(* IEC 61131-3 sources: eCockpitGit/test_project/src/%F%00 Library/%F%Common Functions/%F%Networking, 7 files *)

(* ---- %POU%BASE64Decode.st ---- *)
//This function decodes a base64 string to a normal string or byte array
// |**Version**|**Author**| **Date** |**Changes**
// | 1         | NSN      | 19-05-20 | Creation
FUNCTION BASE64Decode : BOOL
VAR_INPUT
	inStr		:POINTER TO BYTE;
	outStr		:POINTER TO BYTE;		//Out string must be at least 3/4 as long as input string and also a multiple of 4
END_VAR
VAR
	inStrNext	:POINTER TO BYTE := inStr + 1;
	baseBuffer	:BYTE;
END_VAR
VAR CONSTANT
	base64Vars	:ARRAY[43..122] OF BYTE := [62,0,0,0,63,52,53,54,55,56,57,58,59,60,61,0,0,0,0,0,0,0,0,1,2,3,4,5,6,7,8,9,10,11,12,13,14,15,16,17,18,19,20,21,22,23,24,25,0,0,0,0,0,0,26,27,28,29,30,31,32,33,34,35,36,37,38,39,40,41,42,43,44,45,46,47,48,49,50,51];
END_VAR

(*%!%__DELIMITER__%!%*)
WHILE inStr^ <> 0 AND inStrNext^ <> 0 DO
	baseBuffer				:=		SHL(base64Vars[inStr^],2) OR SHR(base64Vars[inStrNext^],4);
	outStr^					:=		baseBuffer;
	inStr					:=		inStr + 1;
	inStrNext				:=		inStr + 1;
	outStr					:=		outStr + 1;
	IF inStr^ <> 0 AND inStrNext^ <> 0 THEN
		baseBuffer			:=		SHL(base64Vars[inStr^],4) OR SHR(base64Vars[inStrNext^],2);
		outStr^				:=		baseBuffer;
		inStr				:=		inStr + 1;
		inStrNext			:=		inStr + 1;
		outStr				:=		outStr + 1;
		IF inStr^ <> 0 AND inStrNext^ <> 0 THEN
			baseBuffer		:=		SHL(base64Vars[inStr^],6) OR base64Vars[inStrNext^];
			outStr^			:=		baseBuffer;
			inStr			:=		inStr + 2;
			inStrNext		:=		inStr + 1;
			outStr			:=		outStr + 1;
		END_IF
	END_IF
END_WHILE

(* ---- %POU%BASE64Encode.st ---- *)
//This function encodes a normal string or byte array to a base 64 string
// |**Version**|**Author**| **Date** |**Changes**
// | 1         | NSN      | 19-05-20 | Creation
FUNCTION BASE64Encode : BOOL
VAR_INPUT
	inStr		:POINTER TO BYTE;		//Input string
	outStr		:POINTER TO BYTE;		//Out string must be at least 1/3 longer than input string and also a multiple of 4
END_VAR
VAR
	inStrLast	:POINTER TO BYTE := inStr;
END_VAR
VAR CONSTANT
	base64Vars	:ARRAY[0..63] OF BYTE := [65,66,67,68,69,70,71,72,73,74,75,76,77,78,79,80,81,82,83,84,85,86,87,88,89,90,97,98,99,100,101,102,103,104,105,106,107,108,109,110,111,112,113,114,115,116,117,118,119,120,121,122,48,49,50,51,52,53,54,55,56,57,43,47];
END_VAR

(*%!%__DELIMITER__%!%*)
WHILE inStr^ <> 0 DO
	outStr^					:=		base64Vars[SHR(inStr^,2)];
	inStrLast				:=		inStr;
	inStr					:=		inStr + 1;
	outStr					:=		outStr + 1;
	IF inStr^ = 0 THEN
		outStr^				:=		base64Vars[SHR(inStr^,4) OR SHL(inStrLast^,4) AND 63];
		outStr				:=		outStr + 1;
		outStr^				:=		EASCII.Equal;
		outStr				:=		outStr + 1;
		outStr^				:=		EASCII.Equal;
	ELSE
		outStr^				:=		base64Vars[SHR(inStr^,4) OR SHL(inStrLast^,4) AND 63];
		inStrLast			:=		inStr;
		outStr				:=		outStr + 1;
		inStr				:=		inStr + 1;
		IF inStr^ = 0 AND inStrLast^ = 0 THEN
			outStr^			:=		EASCII.Equal;
			outStr			:=		outStr + 1;
			outStr^			:=		EASCII.Equal;
		ELSE
			outStr^			:=		base64Vars[SHR(inStr^,6) OR SHL(inStrLast^,2) AND 63];
			outStr			:=		outStr + 1;
			IF inStr^ = 0 THEN
				outStr^		:=		EASCII.Equal;
			ELSE
				outStr^		:=		base64Vars[inStr^ AND 63];
				outStr		:=		outStr + 1;
				inStr		:=		inStr + 1;
			END_IF
		END_IF
	END_IF
END_WHILE
outStr						:=		outStr + 1;
outStr^						:=		0;

(* ---- %POU%BASE64EncodeLen.st ---- *)
//This function encodes a normal string or byte array of fixed lenght to a base 64 string
//This version exists to process strings with zeros in them
// |**Version**|**Author**| **Date** |**Changes**
// | 1         | NSN      | 19-05-20 | Creation
FUNCTION BASE64EncodeLen : BOOL
VAR_INPUT
	inStr		:POINTER TO BYTE;		//Input string
	inLen		:WORD;					//Lenght of input string
	outStr		:POINTER TO BYTE;		//Out string must be at least 1/3 longer than input string and also a multiple of 4
END_VAR
VAR
	inStrLast	:POINTER TO BYTE := inStr;
END_VAR
VAR CONSTANT
	base64Vars	:ARRAY[0..63] OF BYTE := [65,66,67,68,69,70,71,72,73,74,75,76,77,78,79,80,81,82,83,84,85,86,87,88,89,90,97,98,99,100,101,102,103,104,105,106,107,108,109,110,111,112,113,114,115,116,117,118,119,120,121,122,48,49,50,51,52,53,54,55,56,57,43,47];
END_VAR

(*%!%__DELIMITER__%!%*)
WHILE inLen > 0 DO
	outStr^					:=		base64Vars[SHR(inStr^,2)];
	inStrLast				:=		inStr;
	inStr					:=		inStr + 1;
	outStr					:=		outStr + 1;
	inLen					:=		inLen - 1;
	IF inLen = 0 THEN
		outStr^				:=		base64Vars[SHR(0,4) OR SHL(inStrLast^,4) AND 63];
		outStr				:=		outStr + 1;
		outStr^				:=		EASCII.Equal;
		outStr				:=		outStr + 1;
		outStr^				:=		EASCII.Equal;
	ELSE
		outStr^				:=		base64Vars[SHR(inStr^,4) OR SHL(inStrLast^,4) AND 63];
		inStrLast			:=		inStr;
		outStr				:=		outStr + 1;
		inStr				:=		inStr + 1;
		IF inLen = 1 THEN
			outStr^			:=		base64Vars[SHR(0,6) OR SHL(inStrLast^,2) AND 63];
			outStr			:=		outStr + 1;
			outStr^			:=		EASCII.Equal;
			inLen			:=		inLen - 1;
		ELSE
			outStr^			:=		base64Vars[SHR(inStr^,6) OR SHL(inStrLast^,2) AND 63];
			outStr			:=		outStr + 1;
			inLen			:=		inLen - 1;
			IF inLen = 0 THEN
				outStr^		:=		EASCII.Equal;
			ELSE
				outStr^		:=		base64Vars[inStr^ AND 63];
				outStr		:=		outStr + 1;
				inStr		:=		inStr + 1;
				inLen		:=		inLen - 1;
			END_IF
		END_IF
	END_IF
END_WHILE
outStr						:=		outStr + 1;
outStr^						:=		0;

(* ---- %POU%FB_MD5.st ---- *)
//This function block can has a string value
// +-----------+----------+----------+-----------------------------------------------------------------------------------------------------------------------+
// |**Version**|**Author**| **Date** |**Changes**                                                                                                            |
// +-----------+----------+----------+-----------------------------------------------------------------------------------------------------------------------+
// | 1         | NSN      | xx-xx-xx | Creation                                                                                                              |
// +-----------+----------+----------+-----------------------------------------------------------------------------------------------------------------------+
FUNCTION_BLOCK FB_MD5
VAR_INPUT
	sSecret						:STRING;
END_VAR
VAR_OUTPUT
	sMD5						:STRING;
END_VAR
VAR
	abDigest					:ARRAY[0..15] OF BYTE;		//MD5 digest
END_VAR
VAR CONSTANT
	udiNumberOfBytePerSegment	:UDINT := 64;	//higher value -> more time for calculation per PLC-cycle and less PLC cycles are needed for calculation
END_VAR
VAR
	pMemoryBlock				:DWORD; 	//address of memory block
	udiNumberOfBytes			:UDINT; 	//number of bytes of memory block
	wState						:UINT; 		//Statemashine
	udiNumberOfBytesTotal		:UDINT;
	uiLoop						:UINT;
	udiNumberOfBytesUpdated		:UDINT;
	uiNumberOfSegments			:UINT;
//Context
	adwState					:ARRAY[0..3] OF DWORD;
	adwCount					:ARRAY[0..1] OF DWORD;
	abyBuffer					:ARRAY[0..63] OF BYTE;
//Update
	pInput						:POINTER TO BYTE;
	udiLength					:UDINT;
	udiIndex					:UDINT;
	udiPartLen					:UDINT;
	udiInputOffset				:UDINT;
//Final
	Index						:UDINT;
	PadLen						:UDINT;
	abBits						:ARRAY[0..7] OF BYTE;
	abPadding					:ARRAY[0..63] OF BYTE := [16#80];
//Helpers
	bHelp						:BYTE;			//used to calculate the digest
	sHelp						:STRING(2); 	//used to calculate the digest
	pabHelp						:POINTER TO ARRAY [0..255] OF BYTE; //used to add the EndOfString (16#00)
	i							:INT;
END_VAR

(*%!%__DELIMITER__%!%*)
pInput							:=		ADR(sSecret);
udiNumberOfBytesTotal			:=		TO_UDINT(FU_wLenBI(str:=sSecret));
udiNumberOfBytesUpdated			:=		0;
uiNumberOfSegments				:=		0;
adwState[0]						:=		16#67452301;
adwState[1]						:=		16#EFCDAB89;
adwState[2]						:=		16#98BADCFE;
adwState[3]						:=		16#10325476;
adwCount[0]						:=		0;
adwCount[1]						:=		0;
//clear context buffer
FOR uiLoop := 0 TO 63 DO
	abyBuffer[uiLoop]			:=		0 ;
END_FOR
wState							:=		10;

WHILE wState = 10 DO
	IF udiNumberOfBytesUpdated + udiNumberOfBytePerSegment < udiNumberOfBytesTotal THEN
		udiLength				:=		udiNumberOfBytePerSegment;
	ELSE
		udiLength				:=		udiNumberOfBytesTotal - udiNumberOfBytesUpdated;
		wState					:=		20 ;
	END_IF

//MD5 block update operation. Continues an MD5 message-digest operation, processing another message block, and updating the context

	//compute number of bytes MOD 64
	udiIndex					:=		SHR(adwCount[0], 3) AND 16#3F;
	//update number of bits
	adwCount[0]					:=		adwCount[0] + SHL(udiLength,3) ;
	IF adwCount[0] < SHL(udiLength, 3) THEN
		adwCount[1]				:=		adwCount[1] + 1 ;
	END_IF
	adwCount[1]					:=		adwCount[1] + SHR(udiLength, 29);

	udiPartLen					:=		UDINT#64 - udiIndex ;

	//transform as many times as possible
	IF udiLength >= udiPartLen THEN
		MD5_Move(pInput, ADR(abyBuffer[udiIndex]), TO_UINT(udiPartLen));
		MD5_Transform(ADR(adwState),ADR(abyBuffer));
		udiInputOffset			:=		udiPartLen;
		WHILE udiInputOffset + 63 < udiLength DO
			MD5_Transform(ADR(adwState), pInput+udiInputOffset);
			udiInputOffset		:=		udiInputOffset + 64 ;
		END_WHILE ;
		udiIndex				:=		0;
	ELSE
		udiInputOffset			:=		0 ;
	END_IF

	//buffer remaining input
	MD5_Move(pInput+udiInputOffset,ADR(abyBuffer[udiIndex]), TO_UINT(udiLength - udiInputOffset));

	udiNumberOfBytesUpdated		:=		udiNumberOfBytesUpdated + udiLength ;
	uiNumberOfSegments			:=		uiNumberOfSegments + 1;
	pInput						:=		pInput + udiLength;
END_WHILE

//MD5 finalization. Ends an MD5 message-digest operation and writing the the message digest
MD5_Move(ADR(adwCount),ADR(abBits),8);

Index							:=		SHR(adwCount[0], 3) AND 16#3F;
IF Index < 56 THEN
	PadLen						:=		56 - Index ;
ELSE
	PadLen						:=		120 - Index;
END_IF

pInput							:=		ADR(abPadding) ;
udiLength						:=		PadLen ;
//MD5 block update operation. Continues an MD5 message-digest operation, processing another message block, and updating the context.

(* compute number of bytes MOD 64 *)
udiIndex						:=		SHR(adwCount[0], 3) AND 16#3F;
(* update number of bits *)
adwCount[0]						:=		adwCount[0] + SHL(udiLength,3) ;
IF adwCount[0] < SHL(udiLength, 3) THEN
	adwCount[1]					:=		adwCount[1] + 1 ;
END_IF
adwCount[1]						:=		adwCount[1] + SHR(udiLength, 29);

udiPartLen						:=		UDINT#64 - udiIndex ;

//transform as many times as possible.
IF udiLength >= udiPartLen THEN
	MD5_Move(pInput, ADR(abyBuffer[udiIndex]), TO_UINT(udiPartLen));
	MD5_Transform(ADR(adwState),ADR(abyBuffer));
	udiInputOffset				:=		udiPartLen;
	WHILE udiInputOffset + 63 < udiLength DO
		MD5_Transform(ADR(adwState), pInput+udiInputOffset);
		udiInputOffset			:=		udiInputOffset + 64 ;
	END_WHILE ;
	udiIndex					:=		0;
ELSE
	udiInputOffset				:=		0 ;
END_IF

//buffer remaining input
MD5_Move(pInput+udiInputOffset,ADR(abyBuffer[udiIndex]), TO_UINT(udiLength - udiInputOffset));

pInput							:=		ADR(abBits) ;
udiLength						:=		8 ;
//MD5 block update operation. Continues an MD5 message-digest operation, processing another message block, and updating the context.

//compute number of bytes MOD 64
udiIndex						:=		SHR(adwCount[0], 3) AND 16#3F;
//update number of bits
adwCount[0]						:=		adwCount[0] + SHL(udiLength,3) ;
IF adwCount[0] < SHL(udiLength, 3) THEN
	adwCount[1]					:=		adwCount[1] + 1 ;
END_IF
adwCount[1]						:=		adwCount[1] + SHR(udiLength, 29);

udiPartLen						:=		UDINT#64 - udiIndex ;

//transform as many times as possible
IF udiLength >= udiPartLen THEN
	MD5_Move(pInput, ADR(abyBuffer[udiIndex]), TO_UINT(udiPartLen));
	MD5_Transform(ADR(adwState),ADR(abyBuffer));
	udiInputOffset				:=		udiPartLen;
	WHILE udiInputOffset + 63 < udiLength DO
		MD5_Transform(ADR(adwState), pInput+udiInputOffset);
		udiInputOffset			:=		udiInputOffset + 64 ;
	END_WHILE ;
	udiIndex					:=		0;
ELSE
	udiInputOffset				:=		0;
END_IF

//buffer remaining input
MD5_Move(pInput+udiInputOffset,ADR(abyBuffer[udiIndex]), TO_UINT(udiLength - udiInputOffset));

MD5_Move(ADR(adwState), ADR(abDigest) , 16) ;

//Convert the result of the MD5 run from binary to ascii: 16#59 ==> '59' --------
pabHelp							:=		ADR(sMD5);
FOR i := 0 TO 15 DO
	//convert first nibbel
	bHelp						:=		SHR(abDigest[i] AND 16#F0,4);
	IF bHelp <= 9 THEN
		pabHelp^[2*i]			:=		16#30 + bHelp; 		//'0'..'9'
	ELSE
		pabHelp^[2*i]			:=		16#57 + bHelp;  	//'a'..'f'    87+10 = 97 = asc('a')
	END_IF
	//convert second nibbel
	bHelp						:=		abDigest[i] AND 16#0F;
	IF bHelp <= 9 THEN
		pabHelp^[(2*i)+1]		:=		16#30 + bHelp;  	//'0'..'9'
	ELSE
		pabHelp^[(2*i)+1]		:=		16#57 + bHelp;  	//'a'..'f'    87+10 = 97 = asc('a')
	END_IF
END_FOR
pabHelp^[32]					:=		16#00;				//append stringend

(* ---- %POU%FB_SHA1.st ---- *)
//This function calculates sha1 hashes
//First run reset to reset the function block
//Then run input to input the string
//Then run result or resultHex to output the finished hash
// |**Version**|**Author**| **Date** |**Changes**
// | 1         | NSN      | 19-05-20 | Creation
FUNCTION_BLOCK FB_SHA1
VAR
	hash		:ARRAY[0..4] OF DWORD;
	lenLow		:DWORD;
	lenHigh		:DWORD;
	block		:ARRAY[0..63] OF BYTE;
	index		:INT;
	computed	:BOOL;
	corrupted	:BOOL;
END_VAR

(*%!%__DELIMITER__%!%*)

(* ---- %POU%FB_TCPController.st ---- *)
//Controller to simplify TCP connection
// |**Version**|**Author**| **Date** |**Changes**
// | 1         | NSN      | 20-05-22 | Creation
(*	It can be used two ways
	This way has the code directly in the same block as the connection
	IF FB_TCPController.acceptConnection(listener:=TCP.listener) THEN
		//Connection established
	END_IF

	WHILE FB_TCPController.readyToRecieve DO
		Code to handle request
		FB_TCPController.readAmount(amount:=lenght);
	END_WHILE
	FB_TCPController.cycle();

	This way used the message event interface to handle decoding messages
	FB_TCPController.S_message	:=		HandlerForMessages;
	IF FB_TCPController.acceptConnection(listener:=TCP.listener) THEN
		//Connection established
	END_IF

	WHILE FB_TCPController.readyToRecieve DO ; END_WHILE
	FB_TCPController.cycle();
*)

FUNCTION_BLOCK FB_TCPController
VAR_INPUT
	S_index				:WORD;								//Index used to identify controller
	S_management		:ITF_TCPControllerManagement;		//Interface for management events
	S_message			:ITF_TCPControllerMessage;			//Interface for message events
END_VAR
VAR_OUTPUT
	S_open				:BOOL;								//Is true when connection is open
	S_recieveAmount		:DINT;								//How much is left in recieve buffer
END_VAR
VAR
	S_recieveBuffer		:POINTER TO ARRAY[0..99] OF BYTE;	//Reference to recieve buffer
	S_recieveBufferSize	:DINT;								//Size of recieve buffer
	S_sendBuffer		:POINTER TO ARRAY[0..99] OF BYTE;	//Reference to send buffer
	S_sendBufferSize	:DINT;								//Size of send buffer
	S_sendMaxSize		:DINT;								//Estimated max size of sending message, this makes sure that recieved messages are only processed when there is enough space to send the response in the send buffer
	S_maxMessages		:DINT;								//Limit for how many messages can be decoded per cycle
	S_headerSize		:DINT;								//Size of header for tcp message, reading wait until there is at least this amount in the buffer before decoding is performed
	S_stream			:TCP.Stream;
	S_recieveOffset		:DINT;
	S_sendAmount		:DINT;
	S_messageAmount		:DINT;
END_VAR
(*%!%__DELIMITER__%!%*)

(* ---- %POU%FB_TCPMultiPlexer.st ---- *)
//This function block allows for the multiple TCP listeners (eg. multiple network interfaces or ports) to share the same pool of tcp controllers
// |**Version**|**Author**| **Date** |**Changes**
// | 1         | NSN      | 20-05-22 | Creation
(*	It can be used two ways
	This way has the code directly in the same block as the connection
	FB_TCPMultiPlexer.acceptCycle();
	FOR i := 0 to ControllerSize DO
		WHILE FB_TCPController[i].readyToRecieve DO
			Code to handle request
			FB_TCPController[i].readAmount(amount:=lenght);
		END_WHILE
	END_FOR
	FB_TCPMultiPlexer.sendCycle();

	This way used the event interface to decode messages
	FB_TCPMultiPlexer.acceptCycle();
	FB_TCPMultiPlexer.messageCycle();
	FB_TCPMultiPlexer.sendCycle();
*)

FUNCTION_BLOCK FB_TCPMultiPlexer IMPLEMENTS ITF_TCPControllerManagement
VAR_INPUT
	S_management		:ITF_TCPControllerManagement;
END_VAR
VAR_OUTPUT
	S_amountConnected	:WORD;
END_VAR
VAR
	S_messageEvent		:ITF_TCPControllerMessage;
	S_controllers		:POINTER TO ARRAY[0..19] OF FB_TCPController;
	S_controllersSize	:WORD;
	S_listeners			:POINTER TO ARRAY[0..19] OF TCP.Listener;
	S_listenersSize		:WORD;
	S_nextClosed		:WORD;
END_VAR

(*%!%__DELIMITER__%!%*)
